RoboDK station: estacion_practica_tablero.rdk

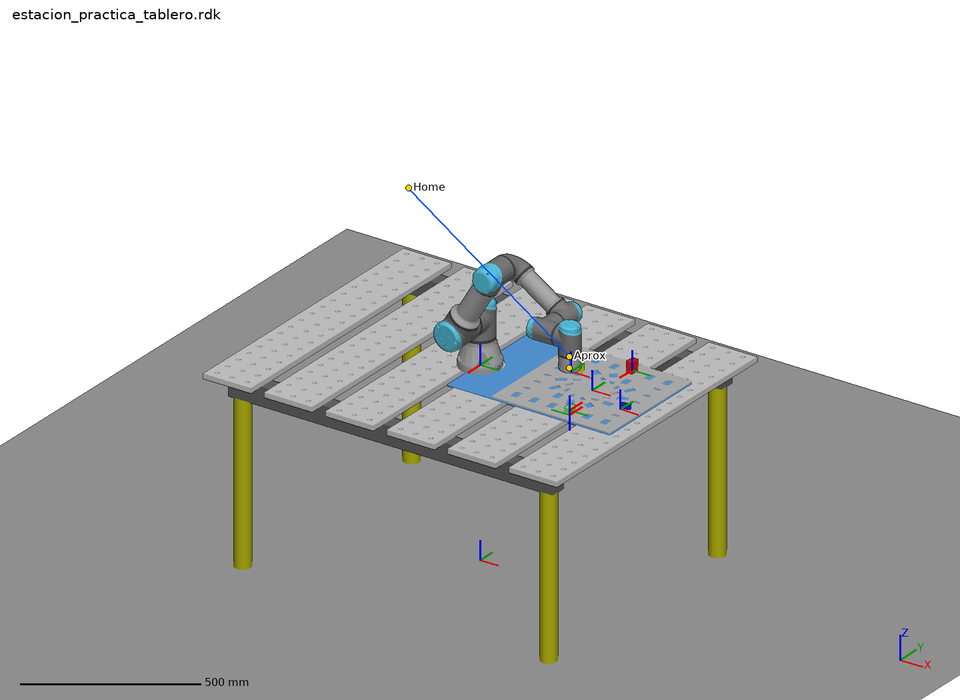
[picture v0: the station drawn from its stored meshes, robots at their saved joint values, targets as dots, program paths as lines]
Station estacion_practica_tablero (saved by RoboDK 5.9.2). Poses are relative to the parent item; angles as X-Y-Z fixed-axis rotations.
  - frame Suelo at (0, 1000, 0) mm
    - object Floor at (0, 0, 0) mm, size 3000 x 3000 x 0 mm, geometry from suelo.sld
    - frame Mesa at (0, 0, 600) mm
      - object Table 1200x1000mm (Welding) at (0, 0, 0) mm, size 1193.8 x 965.2 x 609.6 mm, geometry from mesa.sld
      - frame Base frame at (0, 0, 0) mm
        - object _PIEZA_BaseDeTrabajo at (550, -160, 0) mm, rotated rx 90 ry 0 rz 180 deg, size 550 x 5 x 400 mm, geometry from _PIEZA_BaseDeTrabajo.STL
        - frame workframe at (350, 40, 5) mm
          - object _PIEZA_RebordeBaseDeTrabajoParaBloques at (-200, 200, 0) mm, rotated rx 90 ry 0 rz 0 deg, size 400 x 5 x 400 mm, geometry from _PIEZA_RebordeBaseDeTrabajoParaBloques.STL
        - frame UR3e Base at (0, 0, 0) mm, rotated rx 0 ry 0 rz -90 deg
          - robot UR3e: 6 axes, payload 3 kg, reach 500 mm, repeatability 0.03 mm, weight 11 kg
              modified DH rows (alpha deg, a mm, theta deg, d mm): 0, 0, 0, 151.9; 90, 0, 180, 0; 0, 243.55, 0, 0; 0, 213.2, 0, 131.05; -90, 0, 0, 85.35; 90, 0, 180, 92.1
              joint limits [-360, -360, -360, -360, -360, -360] to [360, 360, 360, 360, 360, 360]; home [0, -90, -90, 0, 90, 0]; saved at [90.818, -121.091, -92.632, -56.277, 90, -179.182]
            - frame TCP at (0, 0, 130) mm
        - frame Pieza1 at (390.28, -125.49, 5) mm, rotated rx 0 ry 0 rz 90 deg
          - object _PIEZA_Bloque20x30x20 at (0, 0, 0) mm, size 30 x 20 x 20 mm, geometry from _PIEZA_Bloque20x30x20.STL
          - target Aprox (Cartesian target) at (0, 0, 180) mm, rotated rx 180 ry 0 rz 0 deg; joints [90.818, -117.022, -88.471, -64.507, 90, -179.182] of UR3e
          - target Target 2 (Cartesian target) at (0, 0, 145) mm, rotated rx 180 ry 0 rz 0 deg; joints [90.818, -121.091, -92.632, -56.277, 90, -179.182] of UR3e
        - frame Pieza2 at (484.19, -14.46, 5) mm
          - object _PIEZA_Bloque20x30x10 at (0, 0, 0) mm, size 30 x 10 x 20 mm, geometry from _PIEZA_Bloque20x30x10.STL
        - frame Pieza3 at (368.96, 206.69, 5) mm, rotated rx 0 ry 0 rz -90.84 deg
          - object _PIEZA_Bloque20x30x40 at (0, 20, 0) mm, rotated rx 90 ry 0 rz 0 deg, size 30 x 40 x 20 mm, geometry from _PIEZA_Bloque20x30x40.STL
        - frame Pieza4 at (251.39, 79, 19.08) mm
          - object _PIEZA_Bloque20x30x30 at (0, 20, 0) mm, rotated rx 90 ry 0 rz 0 deg, size 30 x 30 x 20 mm, geometry from _PIEZA_Bloque20x30x30.STL
    - target Home (joint target) at (-85.35, -223.15, 1208.65) mm, rotated rx 0 ry 90 rz -90 deg; joints [90, -90, 0, 0, 0, 0] of UR3e
  - program Prog1 (5 instructions, listed below)
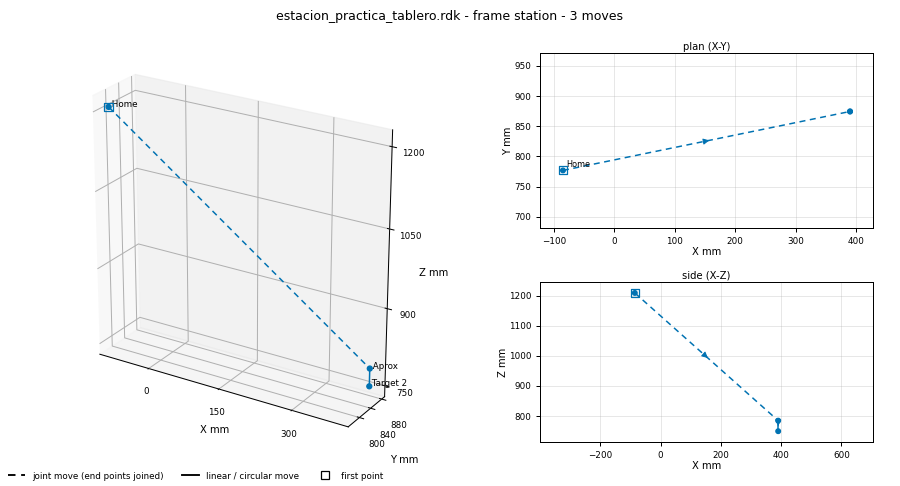
[picture p0: tool path of estacion_practica_tablero.rdk in frame station, 3 of 3 moves have a stored position in this frame; points joined in program order, loops and branches not executed]

--- program Prog1 (robot UR3e) ---
  Est. Ref.: Mesa
  MoveJ (Home)
  Est. Ref.: Pieza1
  MoveJ (Aprox)
  MoveL (Target 2)
